FUNCTION_BLOCK NE_UINT (* IEC 61131-3,Table 28#10 *)
  (* Standard: 61131-3 *)
  (* Version 0.1, 2006-09-14, JHC, Holobloc Inc *)
  (* Compiler header: package fb.rt.plc.comp; *)
  (* Compiler classdef: (IN1 != IN2) *)
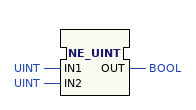
  VAR_INPUT
    IN1 : UINT;
    IN2 : UINT;
  END_VAR
  VAR_OUTPUT
    OUT : BOOL;
  END_VAR
END_FUNCTION_BLOCK
